FUNCTION_BLOCK SM_M2MoveStepsProcedure
VAR_INPUT
	///New state, to be set by the manual implementation
	{attribute 'OPC.UA.DA' := '1'}
	{attribute 'OPC.UA.DA.Access' := '1'}
	state: M2MoveProcedureStates;
	///Actual counter value
	{attribute 'OPC.UA.DA' := '1'}
	{attribute 'OPC.UA.DA.Access' := '1'}
	actualCounterValue AT %I*: UDINT;
	///Number of steps remaining
	{attribute 'OPC.UA.DA' := '1'}
	{attribute 'OPC.UA.DA.Access' := '1'}
	stepsRemaining: UDINT;
END_VAR
VAR_OUTPUT
	///Current status description
	{attribute 'OPC.UA.DA' := '1'}
	{attribute 'OPC.UA.DA.Access' := '1'}
	actualStatus: STRING;
	///Statuses of the state machine
	statuses: M2MoveStepsProcedureStatuses;
END_VAR
VAR_IN_OUT
	{attribute 'OPC.UA.DA' := '0'}
	powerOn: Process;
	{attribute 'OPC.UA.DA' := '0'}
	x: M2XAxis;
	{attribute 'OPC.UA.DA' := '0'}
	y: M2YAxis;
	{attribute 'OPC.UA.DA' := '0'}
	z: M2ZAxis;
	{attribute 'OPC.UA.DA' := '0'}
	tiltX: M2TiltXAxis;
	{attribute 'OPC.UA.DA' := '0'}
	tiltY: M2TiltYAxis;
	{attribute 'OPC.UA.DA' := '0'}
	multiplexer: M2Multiplexer;
	{attribute 'OPC.UA.DA' := '0'}
	config: M2Config;
END_VAR
VAR
END_VAR

statuses.busyStatus( isBusy := NOT((state = M2MoveProcedureStates.IDLE) OR ((state = M2MoveProcedureStates.ABORTED) OR (state = M2MoveProcedureStates.ERROR))) );
statuses.healthStatus(
    isGood := NOT(state = M2MoveProcedureStates.ERROR),
    hasWarning := state = M2MoveProcedureStates.ABORTED);

END_FUNCTION_BLOCK

(* stored: Version 1.1.0.1, ProductVersion 3.1.4019.2
   POU SM_M2MoveStepsProcedure: Id {8c71e008-58be-4e27-adce-805b34ba49bc}, SpecialFunc None *)
